{attribute 'GeneratedUsingTerminal: EL3681-0000-0018'}
{attribute addProperty BoxType "EL3681-0000-0018"}
{attribute addProperty Id "ModeBYTE1RangeSINT1"}
{attribute addProperty CRC "616581440"}
{attribute addProperty Size "2"}
TYPE Settings_24C04940 :
STRUCT
	{attribute addProperty Name "Mode"}
	Mode : BYTE;
	{attribute addProperty Name "Range"}
	Range : SINT;
END_STRUCT
END_TYPE

(* stored: Version 1.2.0.0, ProductVersion 3.1.4024.9
   DUT Settings_24C04940: Id {cc3e2b6e-87dd-4d82-86ec-e84d1cc4883a} *)
